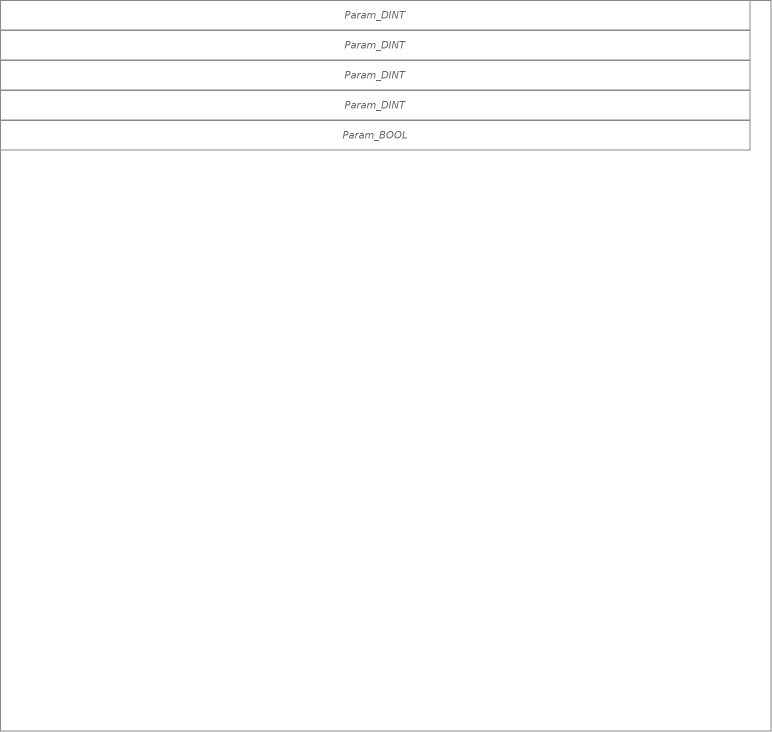
VISUALIZATION Visu_Mparam_General  // 772x732
    Frame (0,120 750x30)
        shows Param_BOOL(nIdx := 6)
    Frame (0,0 750x30)
        shows Param_DINT(nIdx := 3)
    Frame (0,30 750x30)
        shows Param_DINT(nIdx := 4)
    Frame (0,60 750x30)
        shows Param_DINT(nIdx := 5)
    Frame (0,90 750x30)
        shows Param_DINT(nIdx := 6)
    Rectangle (10,690 750x30)
    Rectangle (20,700 750x30)
END_VISUALIZATION

(* stored: Version 1.1.0.1
   Visu Visu_Mparam_General: Id {38861349-9424-4332-bb64-a320fdbe8d36} *)
